Yaskawa INFORM job: s2D_Face_(2).JBI

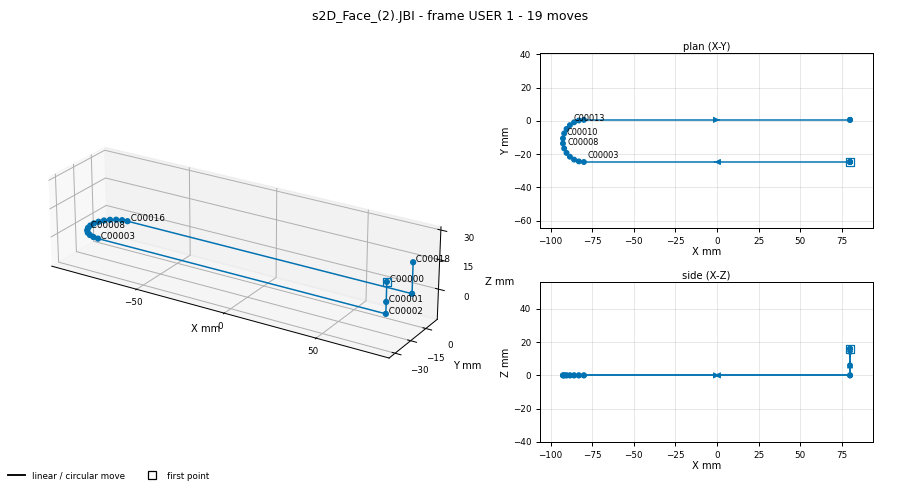
[picture p0: tool path of s2D_Face_(2).JBI in frame USER 1, 19 of 19 moves have a stored position in this frame; points joined in program order, loops and branches not executed]
/JOB
//NAME s2D_Face_(2)
//POS
///NPOS 19,0,0,0,0,0
///USER 1
///TOOL 1
///POSTYPE USER
///RECTAN
///RCONF 1,0,0,0,0,0
C00000=80.000,-24.765,16.000,0.000,-180.000,-30.000
C00001=80.000,-24.765,6.000,0.000,-180.000,-30.000
C00002=80.000,-24.765,0.000,0.000,-180.000,-30.000
C00003=-80.000,-24.765,0.000,0.000,-180.000,-30.000
C00004=-83.032,-24.397,0.000,0.000,-180.000,-30.000
C00005=-85.887,-23.314,0.000,0.000,-180.000,-30.000
C00006=-88.400,-21.579,0.000,0.000,-180.000,-30.000
C00007=-90.425,-19.293,0.000,0.000,-180.000,-30.000
C00008=-91.844,-16.589,0.000,0.000,-180.000,-30.000
C00009=-92.575,-13.624,0.000,0.000,-180.000,-30.000
C00010=-92.575,-10.571,0.000,0.000,-180.000,-30.000
C00011=-91.844,-7.606,0.000,0.000,-180.000,-30.000
C00012=-90.425,-4.902,0.000,0.000,-180.000,-30.000
C00013=-88.400,-2.616,0.000,0.000,-180.000,-30.000
C00014=-85.887,-0.881,0.000,0.000,-180.000,-30.000
C00015=-83.032,0.202,0.000,0.000,-180.000,-30.000
C00016=-80.000,0.570,0.000,0.000,-180.000,-30.000
C00017=80.000,0.570,0.000,0.000,-180.000,-30.000
C00018=80.000,0.570,16.000,0.000,-180.000,-30.000
//INST
///ATTR SC,RW,RJ
////FRAME USER 1
///GROUP1 RB1
///LVARS 2,0,0,0,0,0,0,0
NOP
SET LB000 1
SET LB001 25
MOVJ C00000 VJ=17
MOVL C00001 V=17 PL=LB000 ACC=LB001 DEC=LB001
' Plunge Move Starts
MOVL C00002 V=8 PL=LB000 ACC=LB001 DEC=LB001
' Cutting Move Starts
MOVL C00003 V=17 PL=LB000 ACC=LB001 DEC=LB001
' Link Move Starts
MOVL C00004 V=17 PL=LB000 ACC=LB001 DEC=LB001
MOVL C00005 V=17 PL=LB000 ACC=LB001 DEC=LB001
MOVL C00006 V=17 PL=LB000 ACC=LB001 DEC=LB001
MOVL C00007 V=17 PL=LB000 ACC=LB001 DEC=LB001
MOVL C00008 V=17 PL=LB000 ACC=LB001 DEC=LB001
MOVL C00009 V=17 PL=LB000 ACC=LB001 DEC=LB001
MOVL C00010 V=17 PL=LB000 ACC=LB001 DEC=LB001
MOVL C00011 V=17 PL=LB000 ACC=LB001 DEC=LB001
MOVL C00012 V=17 PL=LB000 ACC=LB001 DEC=LB001
MOVL C00013 V=17 PL=LB000 ACC=LB001 DEC=LB001
MOVL C00014 V=17 PL=LB000 ACC=LB001 DEC=LB001
MOVL C00015 V=17 PL=LB000 ACC=LB001 DEC=LB001
MOVL C00016 V=17 PL=LB000 ACC=LB001 DEC=LB001
' Cutting Move Starts
MOVL C00017 V=17 PL=LB000 ACC=LB001 DEC=LB001
' Rapid Move Starts
MOVL C00018 V=17 PL=LB000 ACC=LB001 DEC=LB001
' By Autodesk Fusion CAM 2.0.20494
' Tool = 1
' Spindle = 5000 RPM
' Set Position Level
' Set Acceleration
' Program Start
' First Toolpath Point
END
